FUNCTION_BLOCK EL2258
VAR
	{attribute addProperty Name "WcState"}
	_wcState : WcStateInputToggle;
	{attribute addProperty Name "Info data"}
	_infoData : InfoDataAdsDC;
	_io : EL2258_Data;
END_VAR

PROPERTY IO : REFERENCE TO EL2258_Data
GET
IO REF= _io;
END_GET
END_PROPERTY

PROPERTY WcState : REFERENCE TO WcStateInputToggle
GET
WcState REF= _wcState;
END_GET
END_PROPERTY

END_FUNCTION_BLOCK

(* stored: Version 1.1.0.1, ProductVersion 3.1.4024.9
   POU EL2258: Id {69fb0ae0-8334-098f-036f-44ca433886d8}, SpecialFunc None
   Property IO: Id {e43135a9-ab61-0e96-38f3-d359750d4295}
   Get Get: Id {b2ae1524-8d1c-01f3-34a8-5cc2ce8eafca}
   Property WcState: Id {edb5fa1b-51bd-01c1-1d95-6270f41fb745}
   Get Get: Id {89068720-cff5-0833-2296-92b8c3228b02} *)
